% RSLogix 500 project I2P Hands-On 4 - Andrew.RSS, saved by version 10.00.00.00 %
PROJECT "ML03A"    % processor: Bul.1763 MicroLogix 1100 Series B %

PROGRAM FILES
  LAD 2   16 rungs

DATA FILES
  O0 OUTPUT  4 elements
  I1 INPUT  6 elements
  S2 STATUS  66 elements
  B3 BINARY  1 elements
  T4 TIMER  1 elements
  C5 COUNTER  1 elements
  R6 CONTROL  1 elements
  N7 INTEGER  1 elements
  F8 FLOAT  1 elements

LADDER 2
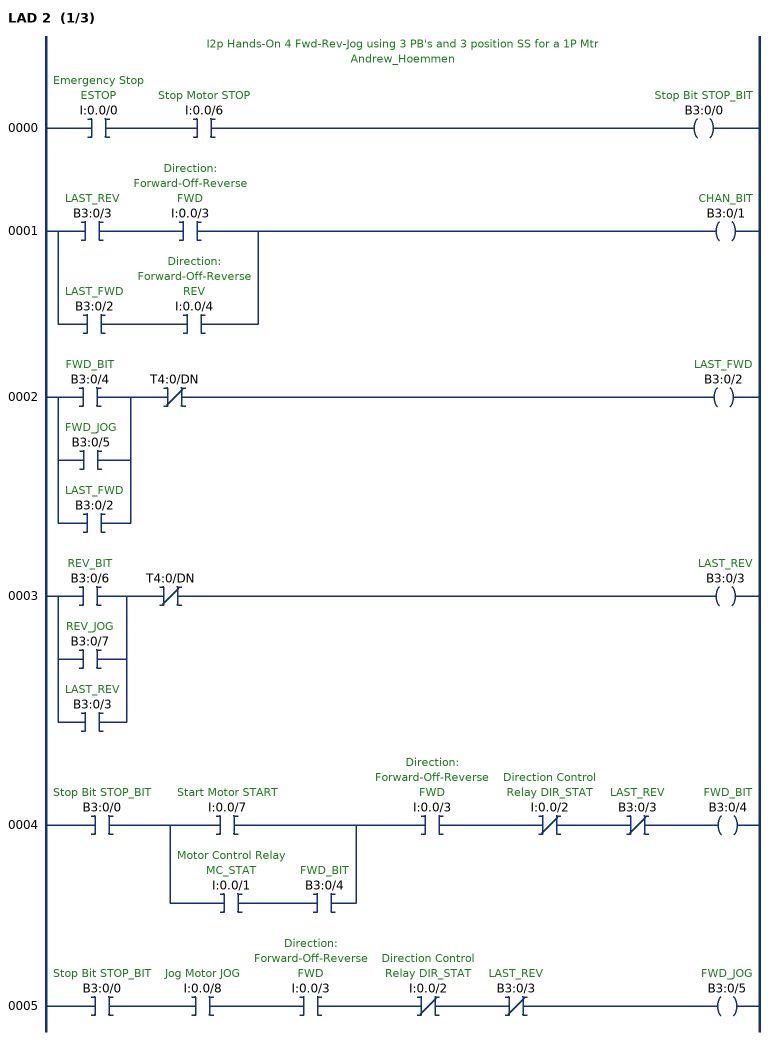
% Rung: 0 %
% I2p Hands-On 4 Fwd-Rev-Jog using 3 PB's and 3 position SS for a 1P Mtr
% Andrew_Hoemmen %
SOR XIC I:0.0/0 XIC I:0.0/6 OTE B3:0/0 EOR
%   I:0.0/0  ESTOP  "Emergency Stop" %
%   I:0.0/6  STOP  "Stop Motor" %
%   B3:0/0  STOP_BIT  "Stop Bit" %
% Rung: 1 %
SOR BST XIC B3:0/3 XIC I:0.0/3 NXB XIC B3:0/2 XIC I:0.0/4 BND OTE B3:0/1 EOR
%   B3:0/3  LAST_REV %
%   I:0.0/3  FWD  "Direction: Forward-Off-Reverse" %
%   B3:0/2  LAST_FWD %
%   I:0.0/4  REV  "Direction: Forward-Off-Reverse" %
%   B3:0/1  CHAN_BIT %
% Rung: 2 %
SOR BST BST XIC B3:0/4 NXB XIC B3:0/5 BND NXB XIC B3:0/2 BND XIO T4:0/DN OTE B3:0/2 EOR
%   B3:0/4  FWD_BIT %
%   B3:0/5  FWD_JOG %
%   B3:0/2  LAST_FWD %
% Rung: 3 %
SOR BST BST XIC B3:0/6 NXB XIC B3:0/7 BND NXB XIC B3:0/3 BND XIO T4:0/DN OTE B3:0/3 EOR
%   B3:0/6  REV_BIT %
%   B3:0/7  REV_JOG %
%   B3:0/3  LAST_REV %
% Rung: 4 %
SOR XIC B3:0/0 BST XIC I:0.0/7 NXB XIC I:0.0/1 XIC B3:0/4 BND XIC I:0.0/3 XIO I:0.0/2 XIO B3:0/3 OTE B3:0/4 EOR
%   B3:0/0  STOP_BIT  "Stop Bit" %
%   I:0.0/7  START  "Start Motor" %
%   I:0.0/1  MC_STAT  "Motor Control Relay" %
%   B3:0/4  FWD_BIT %
%   I:0.0/3  FWD  "Direction: Forward-Off-Reverse" %
%   I:0.0/2  DIR_STAT  "Direction Control Relay" %
%   B3:0/3  LAST_REV %
% Rung: 5 %
SOR XIC B3:0/0 XIC I:0.0/8 XIC I:0.0/3 XIO I:0.0/2 XIO B3:0/3 OTE B3:0/5 EOR
%   B3:0/0  STOP_BIT  "Stop Bit" %
%   I:0.0/8  JOG  "Jog Motor" %
%   I:0.0/3  FWD  "Direction: Forward-Off-Reverse" %
%   I:0.0/2  DIR_STAT  "Direction Control Relay" %
%   B3:0/3  LAST_REV %
%   B3:0/5  FWD_JOG %

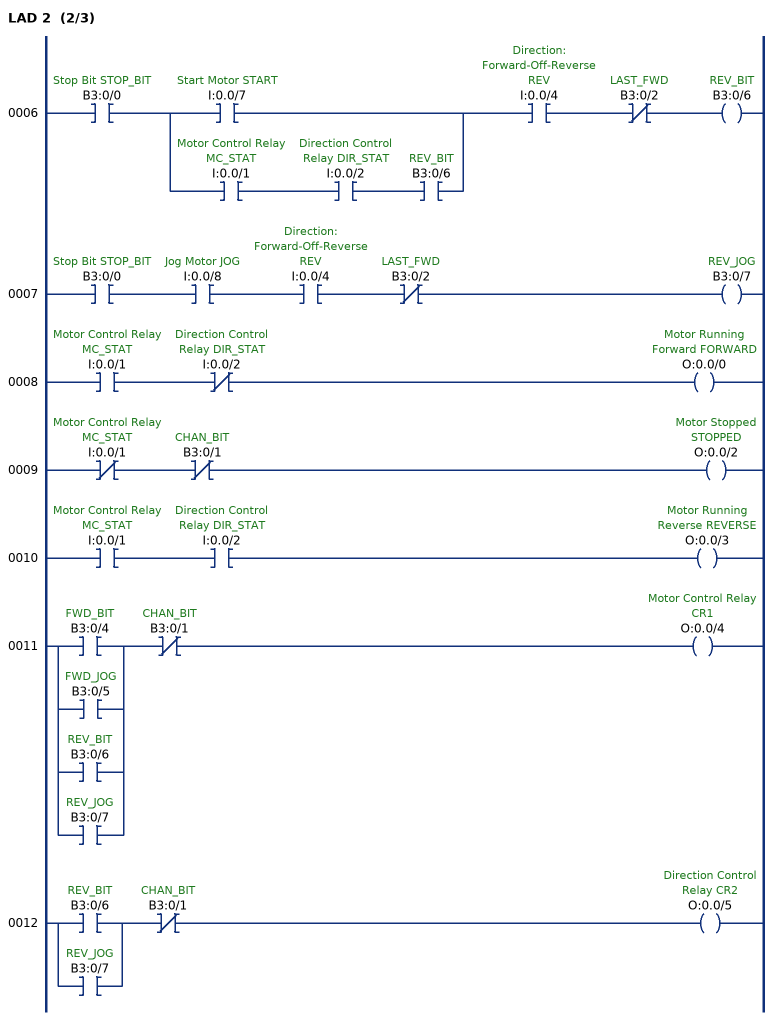
% Rung: 6 %
SOR XIC B3:0/0 BST XIC I:0.0/7 NXB XIC I:0.0/1 XIC I:0.0/2 XIC B3:0/6 BND XIC I:0.0/4 XIO B3:0/2 OTE B3:0/6 EOR
%   B3:0/0  STOP_BIT  "Stop Bit" %
%   I:0.0/7  START  "Start Motor" %
%   I:0.0/1  MC_STAT  "Motor Control Relay" %
%   I:0.0/2  DIR_STAT  "Direction Control Relay" %
%   B3:0/6  REV_BIT %
%   I:0.0/4  REV  "Direction: Forward-Off-Reverse" %
%   B3:0/2  LAST_FWD %
% Rung: 7 %
SOR XIC B3:0/0 XIC I:0.0/8 XIC I:0.0/4 XIO B3:0/2 OTE B3:0/7 EOR
%   B3:0/0  STOP_BIT  "Stop Bit" %
%   I:0.0/8  JOG  "Jog Motor" %
%   I:0.0/4  REV  "Direction: Forward-Off-Reverse" %
%   B3:0/2  LAST_FWD %
%   B3:0/7  REV_JOG %
% Rung: 8 %
SOR XIC I:0.0/1 XIO I:0.0/2 OTE O:0.0/0 EOR
%   I:0.0/1  MC_STAT  "Motor Control Relay" %
%   I:0.0/2  DIR_STAT  "Direction Control Relay" %
%   O:0.0/0  FORWARD  "Motor Running Forward" %
% Rung: 9 %
SOR XIO I:0.0/1 XIO B3:0/1 OTE O:0.0/2 EOR
%   I:0.0/1  MC_STAT  "Motor Control Relay" %
%   B3:0/1  CHAN_BIT %
%   O:0.0/2  STOPPED  "Motor Stopped" %
% Rung: 10 %
SOR XIC I:0.0/1 XIC I:0.0/2 OTE O:0.0/3 EOR
%   I:0.0/1  MC_STAT  "Motor Control Relay" %
%   I:0.0/2  DIR_STAT  "Direction Control Relay" %
%   O:0.0/3  REVERSE  "Motor Running Reverse" %
% Rung: 11 %
SOR BST XIC B3:0/4 NXB BST XIC B3:0/5 NXB BST XIC B3:0/6 NXB XIC B3:0/7 BND BND BND XIO B3:0/1 OTE O:0.0/4 EOR
%   B3:0/4  FWD_BIT %
%   B3:0/5  FWD_JOG %
%   B3:0/6  REV_BIT %
%   B3:0/7  REV_JOG %
%   B3:0/1  CHAN_BIT %
%   O:0.0/4  CR1  "Motor Control Relay" %
% Rung: 12 %
SOR BST XIC B3:0/6 NXB XIC B3:0/7 BND XIO B3:0/1 OTE O:0.0/5 EOR
%   B3:0/6  REV_BIT %
%   B3:0/7  REV_JOG %
%   B3:0/1  CHAN_BIT %
%   O:0.0/5  CR2  "Direction Control Relay" %

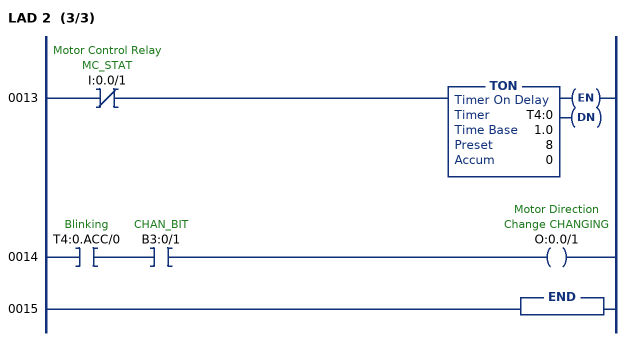
% Rung: 13 %
SOR XIO I:0.0/1 TON T4:0 1.0 8 0 EOR
%   I:0.0/1  MC_STAT  "Motor Control Relay" %
% Rung: 14 %
SOR XIC T4:0.ACC/0 XIC B3:0/1 OTE O:0.0/1 EOR
%   T4:0.ACC/0  "Blinking" %
%   B3:0/1  CHAN_BIT %
%   O:0.0/1  CHANGING  "Motor Direction Change" %
% Rung: 15 %
SOR END EOR

OTHER DOCUMENTED ADDRESSES
  I:0.0/5  2PSS_A  "2p ss,pos.A (up)=ON"

DATA TABLE (non-zero values as saved)
DATA T4
% .PRE .ACC %
% T4:0 % 8 0
